# EPICS IOC start-up script: iocBoot/iocxxx/examples/detectors/ADPointGrey.iocsh
#- INSTANCE  - Used for Camera Port Name and detector pv name
#- ID        - Camera ID
#- XSIZE     - Image Width
#- YSIZE     - Image Height
#- TYPE      - Image Datatype, default: Int8
#- COLORS    - Number of colors, default: 1
#- SUB       - Pointgrey substitutions file, default: examples/detectors/pointGrey.substitutions

epicsEnvSet("EPICS_DB_INCLUDE_PATH", "$(EPICS_DB_INCLUDE_PATH):$(ADCORE)/db:$(ADPOINTGREY)/db")

# pointGreyConfig(const char *portName, int cameraId, int traceMask, int memoryChannel,
#                 int maxBuffers, size_t maxMemory, int priority, int stackSize)
pointGreyConfig("$(INSTANCE)", $(ID), 0x1, 0)

dbLoadRecords("$(ADPOINTGREY)/db/pointGrey.template", "P=$(PREFIX),R=$(INSTANCE):,PORT=$(INSTANCE),ADDR=0,TIMEOUT=1")
dbLoadTemplate("$(SUB=examples/detectors/pointGrey.substitutions)", "P=$(PREFIX),R=$(INSTANCE):,PORT=$(INSTANCE)")

# Create a standard arrays plugin
NDStdArraysConfigure("Image1", 3, 0, "$(INSTANCE)", 0, 2000000)

# Need to determine certain values from input parameters
iocshRun('epicsEnvSet("__FTVL", "$($(TYPE=Int8)_VAL)")', "Int8_VAL=UCHAR, UInt8_VAL=UCHAR, Int16_VAL=SHORT, UInt16_VAL=SHORT, Int32_VAL=LONG, UInt32_VAL=LONG, Float32_VAL=DOUBLE, Float64_VAL=DOUBLE")
iocshRun('epicsEnvSet("__TYPE", "$($(TYPE=Int8)_VAL)")', "Int8_VAL=Int8, UInt8_VAL=Int8, Int16_VAL=Int16, UInt16_VAL=Int16, Int32_VAL=Int32, UInt32_VAL=Int32, Float32_VAL=Float32, Float64_VAL=Float64")
iocshRun('epicsEnvSet("__BYTES", "$($(TYPE=Int8)_VAL)")', "Int8_VAL=1, UInt8_VAL=1, Int16_VAL=2, UInt16_VAL=2, Int32_VAL=4, UInt32_VAL=4, Float32_VAL=4, Float64_VAL=8")
luaCmd("epicsEnvSet('__SIZE', tostring((COLORS*XSIZE*YSIZE)|0))", "COLORS=$(COLORS=1), XSIZE=$(XSIZE), YSIZE=$(YSIZE)")
luaCmd("epicsEnvSet('EPICS_CA_MAX_ARRAY_BYTES', tostring(math.ceil(1.1 * SIZE * BYTES)))", "SIZE=$(__SIZE), BYTES=$(__BYTES)")

dbLoadRecords("$(ADCORE)/ADApp/Db/NDStdArrays.template", "P=$(PREFIX),R=image1:,PORT=Image1,ADDR=0,TIMEOUT=1,NDARRAY_PORT=$(INSTANCE),TYPE=$(__TYPE),FTVL=$(__FTVL),NELEMENTS=$(__SIZE)")

epicsEnvUnset("__FTVL")
epicsEnvUnset("__TYPE")
epicsEnvUnset("__BYTES")
epicsEnvUnset("__SIZE")

iocshLoad("$(ADCORE)/iocBoot/commonPlugins.cmd", "PREFIX=$(PREFIX), PORT=$(INSTANCE), QSIZE=20, XSIZE=$(XSIZE), YSIZE=$(YSIZE), NCHANS=1024, CBUFFS=20, MAX_THREADS=5")

set_requestfile_path("$(ADPOINTGREY)/db")

#- Records with dynamic enums need to be processed again because the enum values are not available during iocInit.
doAfterIocInit("dbpf('$(PREFIX)$(INSTANCE):cam1:Format7Mode.PROC', '1')")
doAfterIocInit("dbpf('$(PREFIX)$(INSTANCE):cam1:PixelFormat.PROC', '1')")

#- Wait for callbacks on the property limits (DRVL, DRVH) to complete
doAfterIocInit("epicsThreadSleep(1.0)")

#- Records that depend on the state of the dynamic enum records or property limits also need to be processed again
#- Other property records may need to be added to this list
doAfterIocInit("dbpf('$(PREFIX)$(INSTANCE):cam1:FrameRate.PROC', '1')")
doAfterIocInit("dbpf('$(PREFIX)$(INSTANCE):cam1:FrameRateValAbs.PROC', '1')")
doAfterIocInit("dbpf('$(PREFIX)$(INSTANCE):cam1:AcquireTime.PROC', '1')")
